FUNCTION_BLOCK Hysteresis
VAR_INPUT
	EN: BOOL := TRUE;
	Value: LREAL;
	LimitValue: LREAL;
	Offset: LREAL; 
END_VAR
VAR_OUTPUT
	ENO: BOOL;
	Above: BOOL;
	Below: BOOL;
END_VAR
VAR
	Hysteresis: INT;
	CurValue: LREAL;
	PreValue: LREAL;
	HystLimit: LREAL;
	HystOffset: LREAL;
END_VAR

HystLimit := LimitValue;
HystOffset := Offset;
IF EN THEN
	Update(Value);
ELSE
	Reset();
END_IF
PreValue := CurValue;
CurValue := Value;
ENO := EN;

METHOD Reset
VAR_INPUT
END_VAR
Hysteresis := 0;
Above := FALSE;
Below := FALSE;
END_METHOD

METHOD PRIVATE Update
VAR_INPUT
	Value: LREAL; 
END_VAR
IF ABS(Value - HystLimit) >= ABS(HystOffset) THEN
	Hysteresis := 0;
END_IF
IF (Value > (LimitValue + Offset * Hysteresis)) AND (PreValue <= (LimitValue + Offset * Hysteresis)) THEN
	IF Hysteresis > -1 THEN
		Hysteresis := Hysteresis - 1;
	END_IF
END_IF
IF (Value <= (LimitValue + Offset * Hysteresis)) AND (PreValue > (LimitValue + Offset * Hysteresis)) THEN
	IF Hysteresis < 1 THEN
		Hysteresis := Hysteresis + 1;
	END_IF
END_IF
Above := CurValue > (LimitValue + HystOffset * Hysteresis);
Below := CurValue <= (LimitValue + HystOffset * Hysteresis);
END_METHOD

END_FUNCTION_BLOCK

(* stored: Version 1.1.0.1, ProductVersion 3.1.4024.3
   POU Hysteresis: Id {d8e65019-ab90-4b7b-9745-c0769a498cb8}, SpecialFunc None
   Method Reset: Id {af996c25-dd0c-4959-adb8-1ed05b4ea3bb}
   Method Update: Id {39d0cef1-d6c8-4060-a19c-158bd1aa1789} *)
